// TIA Portal V17 export
// export: Created 2024-08-26T21:10:48.4510151Z, ExportSetting WithDefaults, DisplayName Totally Integrated Automation Portal, DisplayVersion V17 Update 7, DisplayName TIA Portal Openness, DisplayVersion V17 Update 7, DisplayName TIA Portal Version Control Interface, DisplayVersion V17, DisplayName SINAMICS Startdrive Advanced, DisplayVersion V17 SP2, DisplayName SINAMICS Startdrive G110M, G120, G120C, G120D, G120P, G115D, DisplayVersion V17 SP2, DisplayName SINAMICS Startdrive G130, G150, S120, S150, SINAMICS MV, S210, DisplayVersion V17 SP2, DisplayName STEP 7 Professional, DisplayVersion V17 Update 7, DisplayName STEP 7 Safety, DisplayVersion V17 Update 6, DisplayName WinCC Advanced / Unified PC, DisplayVersion V17 Update 7
FUNCTION "FC_EKS" : Void   // FC305, LAD
TITLE = Euchner Management EKS KEY
{ S7_Optimized_Access := 'FALSE' }
VERSION : 0.1
// stored: AutoNumber false, IsIECCheckEnabled false, SetENOAutomatically false, UDAEnableTagReadback false
   VAR_INPUT
      iKEY_IN : Bool;
      iEKS_LEVEL : Byte;
      iEKS_EMPLOYEE_ID : DWord;
      iEKS_KEY_ID1 : DWord;
      iEKS_KEY_ID2 : DWord;
      iEKS_JOB_FINISHED : Bool;
      "Current_page_of HMI" : Word;
   END_VAR
   VAR_OUTPUT
      qEKS_START_ADDRESS : Byte;
      qEKS_DATA_LENGTH : Byte;
      qEKS_DATA_1 : Byte;
      qEKS_DATA_2 : DWord;
      qEKS_WRITE_CMD : Bool;
   END_VAR
   VAR_TEMP
      tNone : Bool;
      tDBAddressKeys : Int;
      tDBAddressHMIPage : Int;
      tDBKeyStructLength : Int;
      tDBAddress : Int;
      tDBLength : Int;
      tCycle : Int;
      tFill : Int;
      tKey : "udt_EKS_KEY";
      tDBStartAddress : Int;
      tsearch : Bool;
      i : Int;
   END_VAR
   VAR CONSTANT
      DB : Byte := 16#84;
   END_VAR
   VAR_TEMP   // added for the SCL form of the ladder/FBD networks
      _w1 : Bool;
      _w2 : Bool;
   END_VAR
BEGIN

REGION Network 1: Actual HMI page index limits
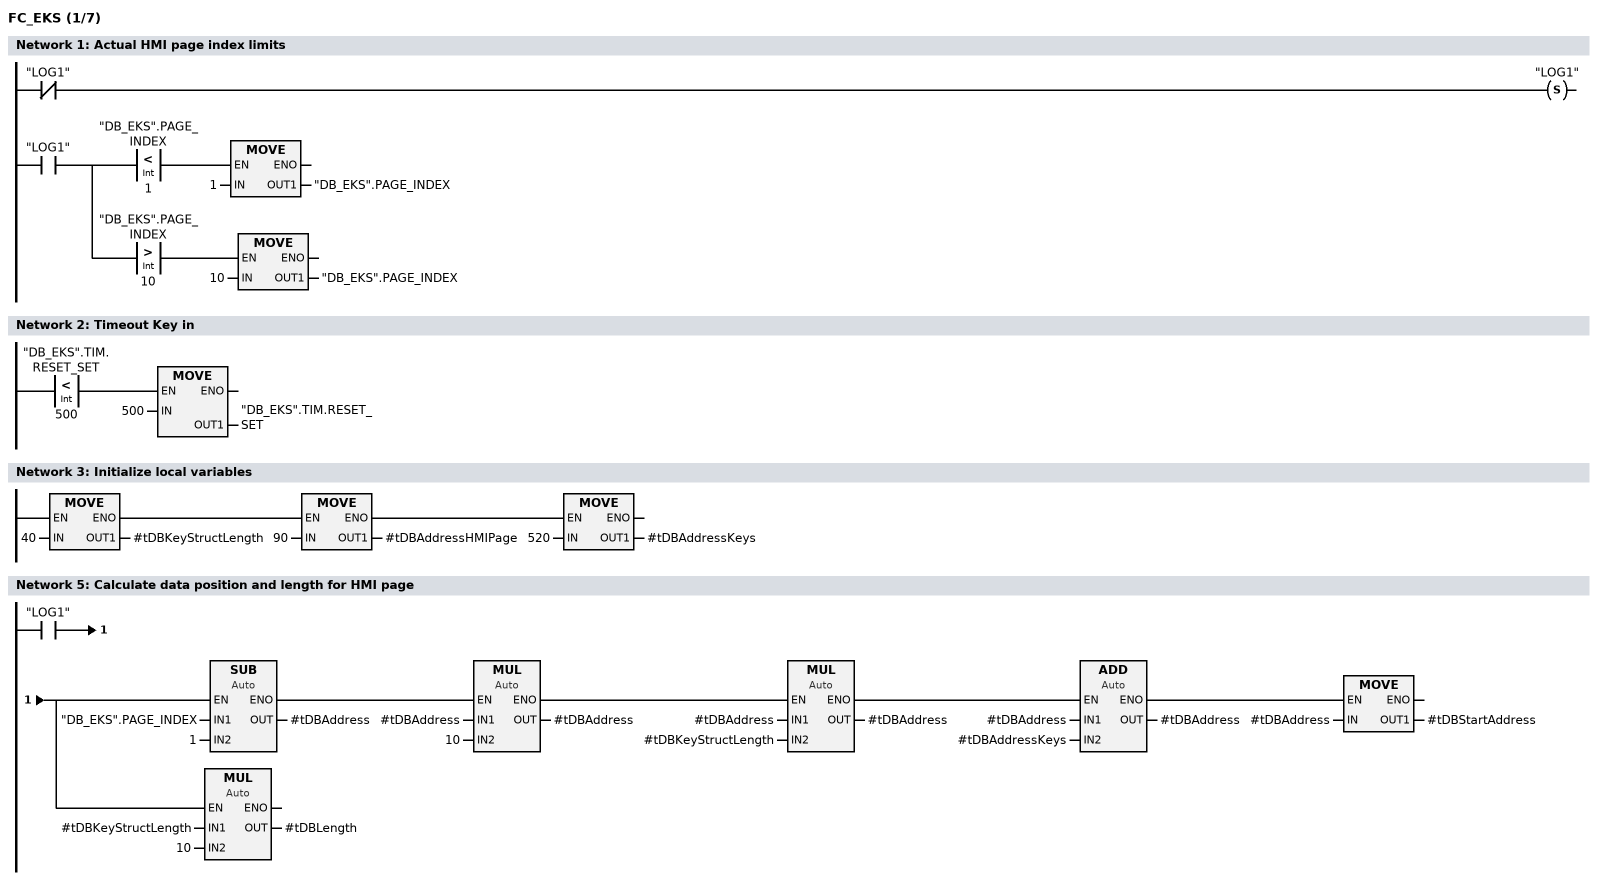
   RUNG wire#powerrail
      I_Contact( "LOG1" )
      S_Coil( "LOG1" )
   END_RUNG
   RUNG wire#powerrail
      Contact( "LOG1" )
      wire#w1
      { S7_Templates := "SrcType := Int" } LT_Contact(in1 := "DB_EKS".PAGE_INDEX, in2 := 1)
      Move(in := 1, out1 => "DB_EKS".PAGE_INDEX)
   END_RUNG
   RUNG wire#w1
      { S7_Templates := "SrcType := Int" } GT_Contact(in1 := "DB_EKS".PAGE_INDEX, in2 := 10)
      Move(in := 10, out1 => "DB_EKS".PAGE_INDEX)
   END_RUNG
   // the same network as SCL:
   IF NOT "LOG1" THEN "LOG1" := TRUE; END_IF;
   IF "LOG1" AND ("DB_EKS".PAGE_INDEX < 1) THEN "DB_EKS".PAGE_INDEX := 1; END_IF;
   IF "LOG1" AND ("DB_EKS".PAGE_INDEX > 10) THEN "DB_EKS".PAGE_INDEX := 10; END_IF;
END_REGION

REGION Network 2: Timeout Key in
   RUNG wire#powerrail
      { S7_Templates := "SrcType := Int" } LT_Contact(in1 := "DB_EKS".TIM.RESET_SET, in2 := 500)
      Move(in := 500, out1 => "DB_EKS".TIM.RESET_SET)
   END_RUNG
   // the same network as SCL:
   IF "DB_EKS".TIM.RESET_SET < 500 THEN "DB_EKS".TIM.RESET_SET := 500; END_IF;
END_REGION

REGION Network 3: Initialize local variables
   RUNG wire#powerrail
      Move(in := 40, out1 => #tDBKeyStructLength)
      Move(in := 90, out1 => #tDBAddressHMIPage)
      Move(in := 520, out1 => #tDBAddressKeys)
   END_RUNG
   // the same network as SCL:
   #tDBKeyStructLength := 40;
   #tDBAddressHMIPage := 90;
   #tDBAddressKeys := 520;
END_REGION

REGION Network 5: Calculate data position and length for HMI page
   RUNG wire#powerrail
      Contact( "LOG1" )
      wire#w1
      Sub(in1 := "DB_EKS".PAGE_INDEX, in2 := 1, out => #tDBAddress)
      Mul(in1 := #tDBAddress, in2 := 10, out => #tDBAddress)
      Mul(in1 := #tDBAddress, in2 := #tDBKeyStructLength, out => #tDBAddress)
      Add(in1 := #tDBAddress, in2 := #tDBAddressKeys, out => #tDBAddress)
      Move(in := #tDBAddress, out1 => #tDBStartAddress)
   END_RUNG
   RUNG wire#w1
      Mul(in1 := #tDBKeyStructLength, in2 := 10, out => #tDBLength)
   END_RUNG
   // the same network as SCL:
   IF "LOG1" THEN
       #tDBAddress := "DB_EKS".PAGE_INDEX - 1;
       #tDBAddress := #tDBAddress * 10;
       #tDBAddress := #tDBAddress * #tDBKeyStructLength;
       #tDBAddress := #tDBAddress + #tDBAddressKeys;
       #tDBStartAddress := #tDBAddress;
       #tDBLength := #tDBKeyStructLength * 10;
   END_IF;
END_REGION

REGION Network 6 (SCL): Copy data for page (10 keys)
   POKE_BLK(area_src:=#DB,
            dbNumber_src:=305,
            byteOffset_src:=#tDBAddress,
            area_dest:=#DB,
            dbNumber_dest:=305,
            byteOffset_dest:=90,
            count:=#tDBLength);
END_REGION

REGION Network 8: Inserted key
   // Store_Key_In is used to display only 1 time the level of euchner during storage function.
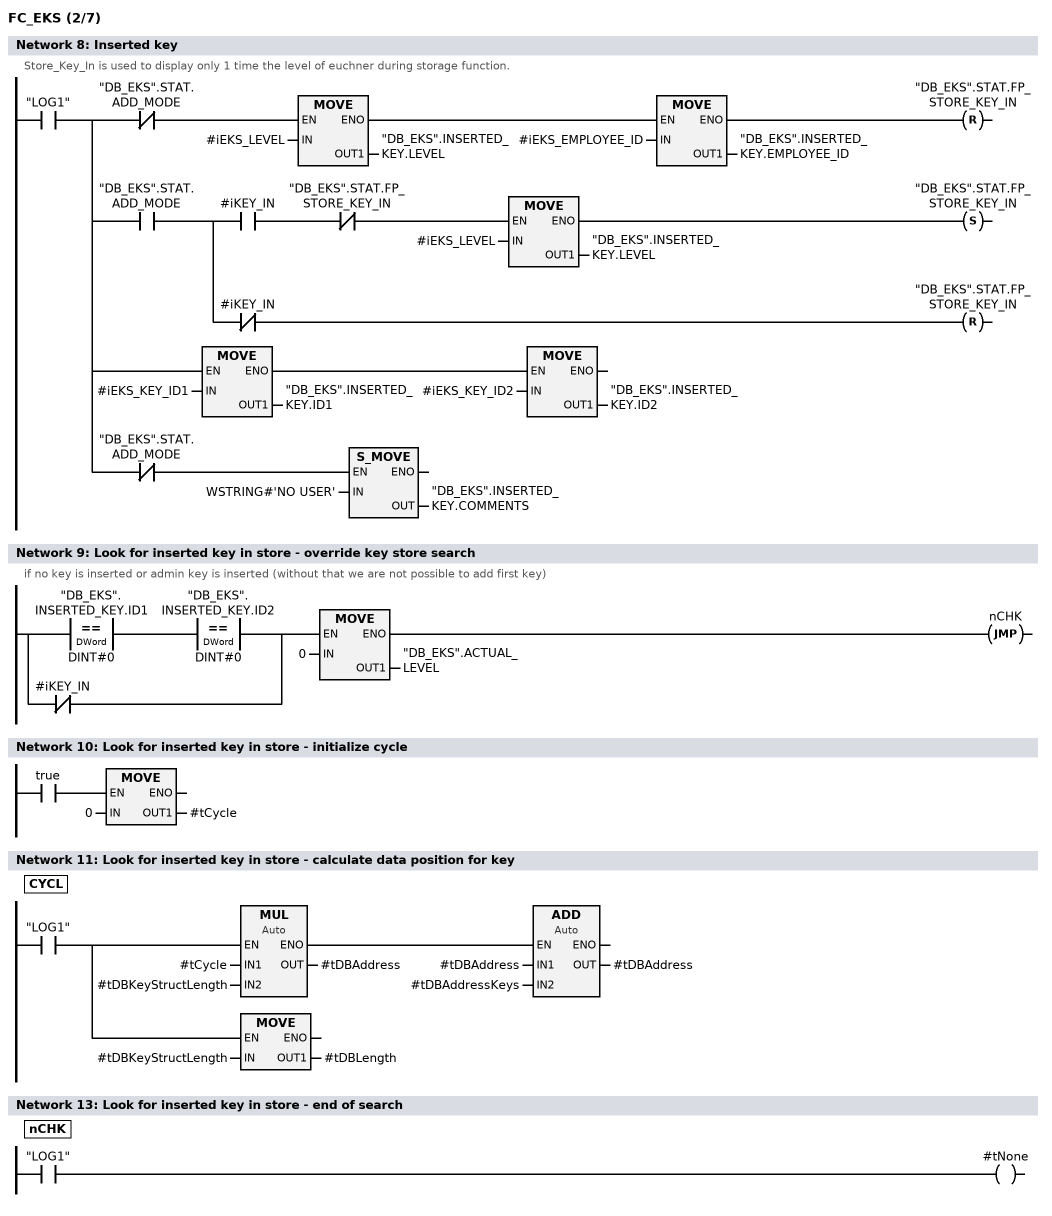
   RUNG wire#powerrail
      Contact( "LOG1" )
      wire#w1
      I_Contact( "DB_EKS".STAT.ADD_MODE )
      Move(in := #iEKS_LEVEL, out1 => "DB_EKS".INSERTED_KEY.LEVEL)
      Move(in := #iEKS_EMPLOYEE_ID, out1 => "DB_EKS".INSERTED_KEY.EMPLOYEE_ID)
      R_Coil( "DB_EKS".STAT.FP_STORE_KEY_IN )
   END_RUNG
   RUNG wire#w1
      Contact( "DB_EKS".STAT.ADD_MODE )
      wire#w2
      Contact( #iKEY_IN )
      I_Contact( "DB_EKS".STAT.FP_STORE_KEY_IN )
      Move(in := #iEKS_LEVEL, out1 => "DB_EKS".INSERTED_KEY.LEVEL)
      S_Coil( "DB_EKS".STAT.FP_STORE_KEY_IN )
   END_RUNG
   RUNG wire#w2
      I_Contact( #iKEY_IN )
      R_Coil( "DB_EKS".STAT.FP_STORE_KEY_IN )
   END_RUNG
   RUNG wire#w1
      Move(in := #iEKS_KEY_ID1, out1 => "DB_EKS".INSERTED_KEY.ID1)
      Move(in := #iEKS_KEY_ID2, out1 => "DB_EKS".INSERTED_KEY.ID2)
   END_RUNG
   RUNG wire#w1
      I_Contact( "DB_EKS".STAT.ADD_MODE )
      S_Move(in := WSTRING#'NO USER', out => "DB_EKS".INSERTED_KEY.COMMENTS)
   END_RUNG
   // the same network as SCL:
   IF "LOG1" AND NOT "DB_EKS".STAT.ADD_MODE THEN
       "DB_EKS".INSERTED_KEY.LEVEL := #iEKS_LEVEL;
       "DB_EKS".INSERTED_KEY.EMPLOYEE_ID := #iEKS_EMPLOYEE_ID;
       "DB_EKS".STAT.FP_STORE_KEY_IN := FALSE;
   END_IF;
   #_w1 := "LOG1" AND "DB_EKS".STAT.ADD_MODE;
   IF #_w1 AND #iKEY_IN AND NOT "DB_EKS".STAT.FP_STORE_KEY_IN THEN
       "DB_EKS".INSERTED_KEY.LEVEL := #iEKS_LEVEL;
       "DB_EKS".STAT.FP_STORE_KEY_IN := TRUE;
   END_IF;
   IF #_w1 AND NOT #iKEY_IN THEN "DB_EKS".STAT.FP_STORE_KEY_IN := FALSE; END_IF;
   IF "LOG1" THEN
       "DB_EKS".INSERTED_KEY.ID1 := #iEKS_KEY_ID1;
       "DB_EKS".INSERTED_KEY.ID2 := #iEKS_KEY_ID2;
   END_IF;
   IF "LOG1" AND NOT "DB_EKS".STAT.ADD_MODE THEN "DB_EKS".INSERTED_KEY.COMMENTS := WSTRING#'NO USER'; END_IF;
END_REGION

REGION Network 9: Look for inserted key in store - override key store search
   // if no key is inserted or admin key is inserted (without that we are not possible to add first key)
   RUNG wire#powerrail
      { S7_Templates := "SrcType := DWord" } EQ_Contact(in1 := "DB_EKS".INSERTED_KEY.ID1, in2 := DINT#0)
      { S7_Templates := "SrcType := DWord" } EQ_Contact(in1 := "DB_EKS".INSERTED_KEY.ID2, in2 := DINT#0)
      wire#w1
      Move(in := 0, out1 => "DB_EKS".ACTUAL_LEVEL)
      JumpCoil( nCHK )
   END_RUNG
   RUNG wire#powerrail
      I_Contact( #iKEY_IN )
   END_RUNG wire#w1
   // the same network as SCL:
   #_w1 := (("DB_EKS".INSERTED_KEY.ID1 = DINT#0) AND ("DB_EKS".INSERTED_KEY.ID2 = DINT#0)) OR NOT #iKEY_IN;
   IF #_w1 THEN
       "DB_EKS".ACTUAL_LEVEL := 0;
       GOTO nCHK;
   END_IF;
END_REGION

REGION Network 10: Look for inserted key in store - initialize cycle
   RUNG wire#powerrail
      Contact( true )
      Move(in := 0, out1 => #tCycle)
   END_RUNG
   // the same network as SCL:
   IF true THEN #tCycle := 0; END_IF;
END_REGION

REGION Network 11: Look for inserted key in store - calculate data position for key
   Label( CYCL )
   RUNG wire#powerrail
      Contact( "LOG1" )
      wire#w1
      Mul(in1 := #tCycle, in2 := #tDBKeyStructLength, out => #tDBAddress)
      Add(in1 := #tDBAddress, in2 := #tDBAddressKeys, out => #tDBAddress)
   END_RUNG
   RUNG wire#w1
      Move(in := #tDBKeyStructLength, out1 => #tDBLength)
   END_RUNG
   // the same network as SCL:
   CYCL:
   IF "LOG1" THEN
       #tDBAddress := #tCycle * #tDBKeyStructLength;
       #tDBAddress := #tDBAddress + #tDBAddressKeys;
       #tDBLength := #tDBKeyStructLength;
   END_IF;
END_REGION

REGION Network 12 (SCL): Look for inserted key in store - check ID of stored key
   FOR #i := 1 TO 130 DO
       #tKey := "DB_EKS".KEYS[#i];
       IF (#tKey.ID1 = "DB_EKS".INSERTED_KEY.ID1) AND
           (#tKey.ID2 = "DB_EKS".INSERTED_KEY.ID2) THEN
           "DB_EKS".ACTUAL_LEVEL := #tKey.LEVEL;
           "DB_EKS".INSERTED_KEY.COMMENTS := #tKey.COMMENTS;
           EXIT;
       END_IF;
   END_FOR;
END_REGION

REGION Network 13: Look for inserted key in store - end of search
   Label( nCHK )
   RUNG wire#powerrail
      Contact( "LOG1" )
      Coil( #tNone )
   END_RUNG
   // the same network as SCL:
   nCHK:
   #tNone := "LOG1";
END_REGION

REGION Network 14: Reset of EKS higher levels until key is removed
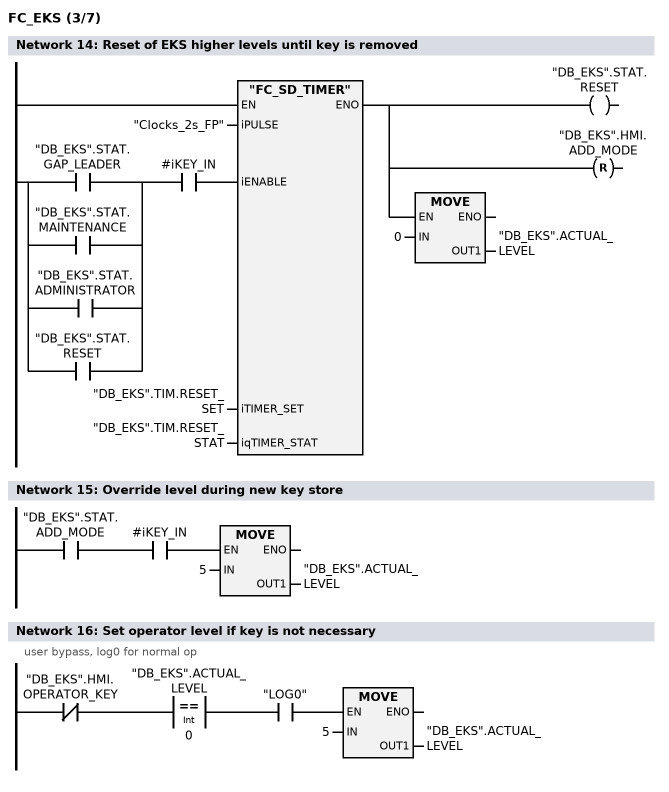
   RUNG wire#powerrail
      "FC_SD_TIMER"(iENABLE := wire#w2, iPULSE := "Clocks_2s_FP", iTIMER_SET := "DB_EKS".TIM.RESET_SET, iqTIMER_STAT := "DB_EKS".TIM.RESET_STAT)
      wire#w3
      Coil( "DB_EKS".STAT.RESET )
   END_RUNG
   RUNG wire#powerrail
      Contact( "DB_EKS".STAT.GAP_LEADER )
      wire#w1
      Contact( #iKEY_IN )
   END_RUNG wire#w2
   RUNG wire#powerrail
      Contact( "DB_EKS".STAT.MAINTENANCE )
   END_RUNG wire#w1
   RUNG wire#powerrail
      Contact( "DB_EKS".STAT.ADMINISTRATOR )
   END_RUNG wire#w1
   RUNG wire#powerrail
      Contact( "DB_EKS".STAT.RESET )
   END_RUNG wire#w1
   RUNG wire#w3
      R_Coil( "DB_EKS".HMI.ADD_MODE )
   END_RUNG
   RUNG wire#w3
      Move(in := 0, out1 => "DB_EKS".ACTUAL_LEVEL)
   END_RUNG
   // the same network as SCL:
   "FC_SD_TIMER"(iPULSE := "Clocks_2s_FP",
                 iENABLE := ("DB_EKS".STAT.GAP_LEADER OR "DB_EKS".STAT.MAINTENANCE OR "DB_EKS".STAT.ADMINISTRATOR OR "DB_EKS".STAT.RESET) AND #iKEY_IN,
                 iTIMER_SET := "DB_EKS".TIM.RESET_SET,
                 iqTIMER_STAT := "DB_EKS".TIM.RESET_STAT,
                 ENO => #_w1);
   "DB_EKS".STAT.RESET := #_w1;
   IF #_w1 THEN
       "DB_EKS".HMI.ADD_MODE := FALSE;
       "DB_EKS".ACTUAL_LEVEL := 0;
   END_IF;
END_REGION

REGION Network 15: Override level during new key store
   RUNG wire#powerrail
      Contact( "DB_EKS".STAT.ADD_MODE )
      Contact( #iKEY_IN )
      Move(in := 5, out1 => "DB_EKS".ACTUAL_LEVEL)
   END_RUNG
   // the same network as SCL:
   IF "DB_EKS".STAT.ADD_MODE AND #iKEY_IN THEN "DB_EKS".ACTUAL_LEVEL := 5; END_IF;
END_REGION

REGION Network 16: Set operator level if key is not necessary
   // user bypass, log0 for normal op
   RUNG wire#powerrail
      I_Contact( "DB_EKS".HMI.OPERATOR_KEY )
      { S7_Templates := "SrcType := Int" } EQ_Contact(in1 := "DB_EKS".ACTUAL_LEVEL, in2 := 0)
      Contact( "LOG0" )
      Move(in := 5, out1 => "DB_EKS".ACTUAL_LEVEL)
   END_RUNG
   // the same network as SCL:
   IF NOT "DB_EKS".HMI.OPERATOR_KEY AND ("DB_EKS".ACTUAL_LEVEL = 0) AND "LOG0" THEN
       "DB_EKS".ACTUAL_LEVEL := 5;
   END_IF;
END_REGION

REGION Network 17: EKS levels
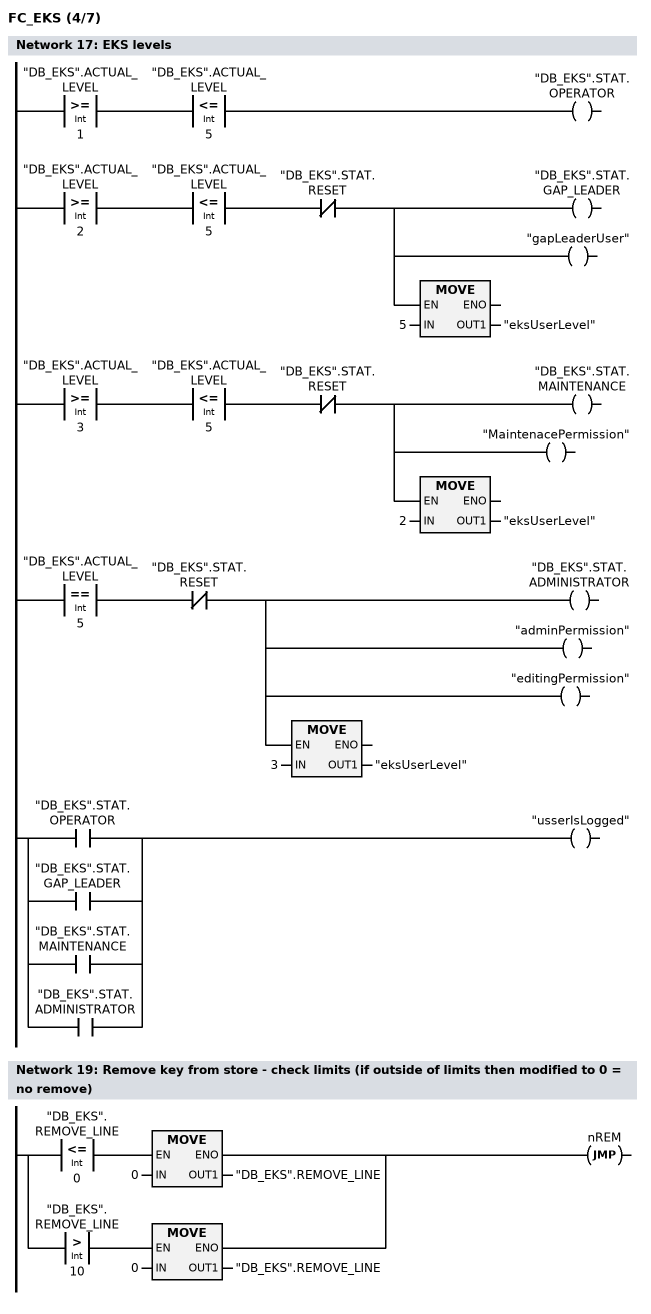
   RUNG wire#powerrail
      { S7_Templates := "SrcType := Int" } GE_Contact(in1 := "DB_EKS".ACTUAL_LEVEL, in2 := 1)
      { S7_Templates := "SrcType := Int" } LE_Contact(in1 := "DB_EKS".ACTUAL_LEVEL, in2 := 5)
      Coil( "DB_EKS".STAT.OPERATOR )
   END_RUNG
   RUNG wire#powerrail
      { S7_Templates := "SrcType := Int" } GE_Contact(in1 := "DB_EKS".ACTUAL_LEVEL, in2 := 2)
      { S7_Templates := "SrcType := Int" } LE_Contact(in1 := "DB_EKS".ACTUAL_LEVEL, in2 := 5)
      I_Contact( "DB_EKS".STAT.RESET )
      wire#w1
      Coil( "DB_EKS".STAT.GAP_LEADER )
   END_RUNG
   RUNG wire#w1
      Coil( "gapLeaderUser" )
   END_RUNG
   RUNG wire#w1
      Move(in := 5, out1 => "eksUserLevel")
   END_RUNG
   RUNG wire#powerrail
      { S7_Templates := "SrcType := Int" } GE_Contact(in1 := "DB_EKS".ACTUAL_LEVEL, in2 := 3)
      { S7_Templates := "SrcType := Int" } LE_Contact(in1 := "DB_EKS".ACTUAL_LEVEL, in2 := 5)
      I_Contact( "DB_EKS".STAT.RESET )
      wire#w2
      Coil( "DB_EKS".STAT.MAINTENANCE )
   END_RUNG
   RUNG wire#w2
      Coil( "MaintenacePermission" )
   END_RUNG
   RUNG wire#w2
      Move(in := 2, out1 => "eksUserLevel")
   END_RUNG
   RUNG wire#powerrail
      { S7_Templates := "SrcType := Int" } EQ_Contact(in1 := "DB_EKS".ACTUAL_LEVEL, in2 := 5)
      I_Contact( "DB_EKS".STAT.RESET )
      wire#w3
      Coil( "DB_EKS".STAT.ADMINISTRATOR )
   END_RUNG
   RUNG wire#w3
      Coil( "adminPermission" )
   END_RUNG
   RUNG wire#w3
      Coil( "editingPermission" )
   END_RUNG
   RUNG wire#w3
      Move(in := 3, out1 => "eksUserLevel")
   END_RUNG
   RUNG wire#powerrail
      Contact( "DB_EKS".STAT.OPERATOR )
      wire#w4
      Coil( "usserIsLogged" )
   END_RUNG
   RUNG wire#powerrail
      Contact( "DB_EKS".STAT.GAP_LEADER )
   END_RUNG wire#w4
   RUNG wire#powerrail
      Contact( "DB_EKS".STAT.MAINTENANCE )
   END_RUNG wire#w4
   RUNG wire#powerrail
      Contact( "DB_EKS".STAT.ADMINISTRATOR )
   END_RUNG wire#w4
   // the same network as SCL:
   "DB_EKS".STAT.OPERATOR := ("DB_EKS".ACTUAL_LEVEL >= 1) AND ("DB_EKS".ACTUAL_LEVEL <= 5);
   "DB_EKS".STAT.GAP_LEADER := ("DB_EKS".ACTUAL_LEVEL >= 2) AND ("DB_EKS".ACTUAL_LEVEL <= 5) AND NOT "DB_EKS".STAT.RESET;
   "gapLeaderUser" := "DB_EKS".STAT.GAP_LEADER;
   IF "DB_EKS".STAT.GAP_LEADER THEN "eksUserLevel" := 5; END_IF;
   "DB_EKS".STAT.MAINTENANCE := ("DB_EKS".ACTUAL_LEVEL >= 3) AND ("DB_EKS".ACTUAL_LEVEL <= 5) AND NOT "DB_EKS".STAT.RESET;
   "MaintenacePermission" := "DB_EKS".STAT.MAINTENANCE;
   IF "DB_EKS".STAT.MAINTENANCE THEN "eksUserLevel" := 2; END_IF;
   "DB_EKS".STAT.ADMINISTRATOR := ("DB_EKS".ACTUAL_LEVEL = 5) AND NOT "DB_EKS".STAT.RESET;
   "adminPermission" := "DB_EKS".STAT.ADMINISTRATOR;
   "editingPermission" := "DB_EKS".STAT.ADMINISTRATOR;
   IF "DB_EKS".STAT.ADMINISTRATOR THEN "eksUserLevel" := 3; END_IF;
   "usserIsLogged" := "DB_EKS".STAT.OPERATOR OR "DB_EKS".STAT.GAP_LEADER OR "DB_EKS".STAT.MAINTENANCE OR "DB_EKS".STAT.ADMINISTRATOR;
END_REGION

REGION Network 19: Remove key from store - check limits (if outside of limits then modified to 0 = no remove)
   RUNG wire#powerrail
      { S7_Templates := "SrcType := Int" } LE_Contact(in1 := "DB_EKS".REMOVE_LINE, in2 := 0)
      Move(in := 0, out1 => "DB_EKS".REMOVE_LINE)
      wire#w1
      JumpCoil( nREM )
   END_RUNG
   RUNG wire#powerrail
      { S7_Templates := "SrcType := Int" } GT_Contact(in1 := "DB_EKS".REMOVE_LINE, in2 := 10)
      Move(in := 0, out1 => "DB_EKS".REMOVE_LINE)
   END_RUNG wire#w1
   // the same network as SCL:
   #_w1 := "DB_EKS".REMOVE_LINE <= 0;
   IF #_w1 THEN "DB_EKS".REMOVE_LINE := 0; END_IF;
   #_w2 := "DB_EKS".REMOVE_LINE > 10;
   IF #_w2 THEN "DB_EKS".REMOVE_LINE := 0; END_IF;
   IF #_w1 OR #_w2 THEN GOTO nREM; END_IF;
END_REGION

REGION Network 20: Remove key from store - calculate data position and length for HMI page
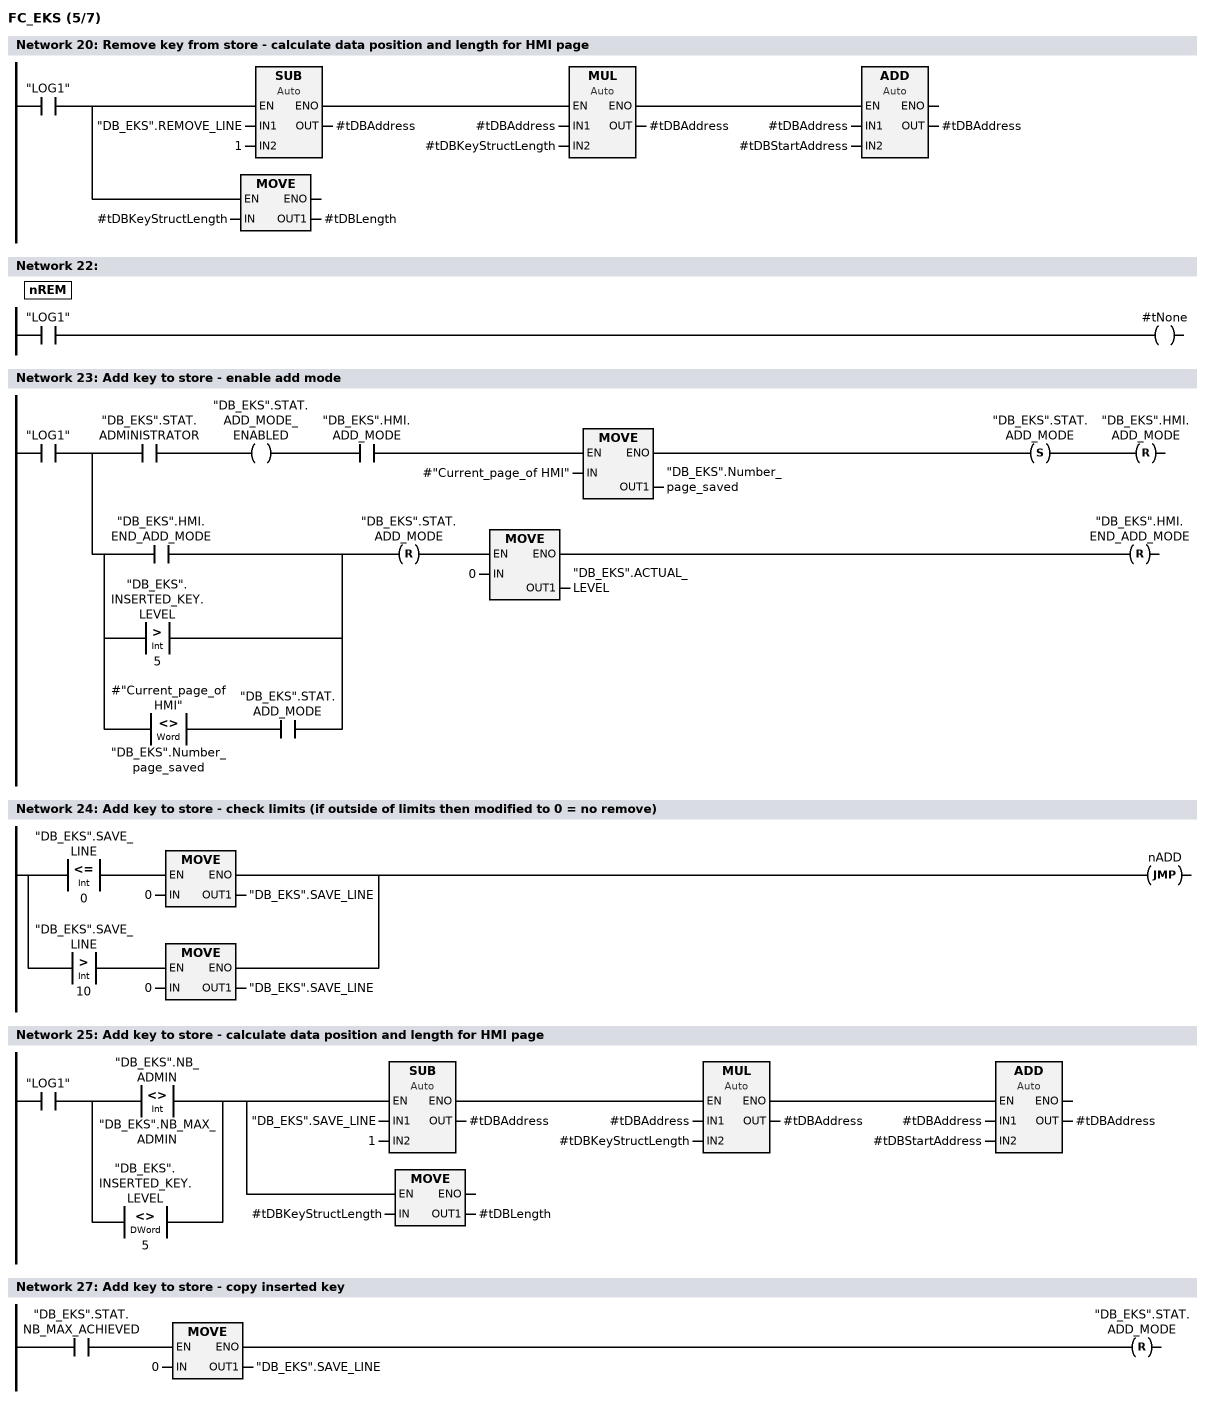
   RUNG wire#powerrail
      Contact( "LOG1" )
      wire#w1
      Sub(in1 := "DB_EKS".REMOVE_LINE, in2 := 1, out => #tDBAddress)
      Mul(in1 := #tDBAddress, in2 := #tDBKeyStructLength, out => #tDBAddress)
      Add(in1 := #tDBAddress, in2 := #tDBStartAddress, out => #tDBAddress)
   END_RUNG
   RUNG wire#w1
      Move(in := #tDBKeyStructLength, out1 => #tDBLength)
   END_RUNG
   // the same network as SCL:
   IF "LOG1" THEN
       #tDBAddress := "DB_EKS".REMOVE_LINE - 1;
       #tDBAddress := #tDBAddress * #tDBKeyStructLength;
       #tDBAddress := #tDBAddress + #tDBStartAddress;
       #tDBLength := #tDBKeyStructLength;
   END_IF;
END_REGION

REGION Network 21 (SCL): Remove key from store - delete key
   #tFill := 0;

   POKE_BLK(area_src:=#DB,
            dbNumber_src:=305,
            byteOffset_src:=5720,
            area_dest:=#DB,
            dbNumber_dest:=305,
            byteOffset_dest:=#tDBAddress,
            count:=#tDBLength);

   "DB_EKS".REMOVE_LINE := 0;
END_REGION

REGION Network 22
   Label( nREM )
   RUNG wire#powerrail
      Contact( "LOG1" )
      Coil( #tNone )
   END_RUNG
   // the same network as SCL:
   nREM:
   #tNone := "LOG1";
END_REGION

REGION Network 23: Add key to store - enable add mode
   RUNG wire#powerrail
      Contact( "LOG1" )
      wire#w1
      Contact( "DB_EKS".STAT.ADMINISTRATOR )
      Coil( "DB_EKS".STAT.ADD_MODE_ENABLED )
      Contact( "DB_EKS".HMI.ADD_MODE )
      Move(in := #"Current_page_of HMI", out1 => "DB_EKS".Number_page_saved)
      S_Coil( "DB_EKS".STAT.ADD_MODE )
      R_Coil( "DB_EKS".HMI.ADD_MODE )
   END_RUNG
   RUNG wire#w1
      Contact( "DB_EKS".HMI.END_ADD_MODE )
      wire#w2
      R_Coil( "DB_EKS".STAT.ADD_MODE )
      Move(in := 0, out1 => "DB_EKS".ACTUAL_LEVEL)
      R_Coil( "DB_EKS".HMI.END_ADD_MODE )
   END_RUNG
   RUNG wire#w1
      { S7_Templates := "SrcType := Int" } GT_Contact(in1 := "DB_EKS".INSERTED_KEY.LEVEL, in2 := 5)
   END_RUNG wire#w2
   RUNG wire#w1
      { S7_Templates := "SrcType := Word" } NE_Contact(in1 := #"Current_page_of HMI", in2 := "DB_EKS".Number_page_saved)
      Contact( "DB_EKS".STAT.ADD_MODE )
   END_RUNG wire#w2
   // the same network as SCL:
   "DB_EKS".STAT.ADD_MODE_ENABLED := "LOG1" AND "DB_EKS".STAT.ADMINISTRATOR;
   IF "DB_EKS".STAT.ADD_MODE_ENABLED AND "DB_EKS".HMI.ADD_MODE THEN
       "DB_EKS".Number_page_saved := #"Current_page_of HMI";
       "DB_EKS".STAT.ADD_MODE := TRUE;
       "DB_EKS".HMI.ADD_MODE := FALSE;
   END_IF;
   #_w1 := "LOG1" AND ("DB_EKS".HMI.END_ADD_MODE OR ("DB_EKS".INSERTED_KEY.LEVEL > 5) OR ((#"Current_page_of HMI" <> "DB_EKS".Number_page_saved) AND "DB_EKS".STAT.ADD_MODE));
   IF #_w1 THEN
       "DB_EKS".STAT.ADD_MODE := FALSE;
       "DB_EKS".ACTUAL_LEVEL := 0;
       "DB_EKS".HMI.END_ADD_MODE := FALSE;
   END_IF;
END_REGION

REGION Network 24: Add key to store - check limits (if outside of limits then modified to 0 = no remove)
   RUNG wire#powerrail
      { S7_Templates := "SrcType := Int" } LE_Contact(in1 := "DB_EKS".SAVE_LINE, in2 := 0)
      Move(in := 0, out1 => "DB_EKS".SAVE_LINE)
      wire#w1
      JumpCoil( nADD )
   END_RUNG
   RUNG wire#powerrail
      { S7_Templates := "SrcType := Int" } GT_Contact(in1 := "DB_EKS".SAVE_LINE, in2 := 10)
      Move(in := 0, out1 => "DB_EKS".SAVE_LINE)
   END_RUNG wire#w1
   // the same network as SCL:
   #_w1 := "DB_EKS".SAVE_LINE <= 0;
   IF #_w1 THEN "DB_EKS".SAVE_LINE := 0; END_IF;
   #_w2 := "DB_EKS".SAVE_LINE > 10;
   IF #_w2 THEN "DB_EKS".SAVE_LINE := 0; END_IF;
   IF #_w1 OR #_w2 THEN GOTO nADD; END_IF;
END_REGION

REGION Network 25: Add key to store - calculate data position and length for HMI page
   RUNG wire#powerrail
      Contact( "LOG1" )
      wire#w1
      { S7_Templates := "SrcType := Int" } NE_Contact(in1 := "DB_EKS".NB_ADMIN, in2 := "DB_EKS".NB_MAX_ADMIN)
      wire#w2
      Sub(in1 := "DB_EKS".SAVE_LINE, in2 := 1, out => #tDBAddress)
      Mul(in1 := #tDBAddress, in2 := #tDBKeyStructLength, out => #tDBAddress)
      Add(in1 := #tDBAddress, in2 := #tDBStartAddress, out => #tDBAddress)
   END_RUNG
   RUNG wire#w1
      { S7_Templates := "SrcType := DWord" } NE_Contact(in1 := "DB_EKS".INSERTED_KEY.LEVEL, in2 := 5)
   END_RUNG wire#w2
   RUNG wire#w2
      Move(in := #tDBKeyStructLength, out1 => #tDBLength)
   END_RUNG
   // the same network as SCL:
   IF "LOG1" AND (("DB_EKS".NB_ADMIN <> "DB_EKS".NB_MAX_ADMIN) OR ("DB_EKS".INSERTED_KEY.LEVEL <> 5)) THEN
       #tDBAddress := "DB_EKS".SAVE_LINE - 1;
       #tDBAddress := #tDBAddress * #tDBKeyStructLength;
       #tDBAddress := #tDBAddress + #tDBStartAddress;
       #tDBLength := #tDBKeyStructLength;
   END_IF;
END_REGION

REGION Network 26 (SCL): Add key to store - copy inserted key
   IF ("DB_EKS".INSERTED_KEY.LEVEL = 5  & NOT "DB_EKS".STAT.NB_MAX_ACHIEVED) OR
       ("DB_EKS".INSERTED_KEY.LEVEL <> 5) THEN
       POKE_BLK(area_src := #DB,
                dbNumber_src := 305,
                byteOffset_src := 50,
                area_dest := #DB,
                dbNumber_dest := 305,
                byteOffset_dest := #tDBAddress,
                count := #tDBLength);
      "DB_EKS".SAVE_LINE := 0;
   END_IF;
END_REGION

REGION Network 27: Add key to store - copy inserted key
   RUNG wire#powerrail
      Contact( "DB_EKS".STAT.NB_MAX_ACHIEVED )
      Move(in := 0, out1 => "DB_EKS".SAVE_LINE)
      R_Coil( "DB_EKS".STAT.ADD_MODE )
   END_RUNG
   // the same network as SCL:
   IF "DB_EKS".STAT.NB_MAX_ACHIEVED THEN
       "DB_EKS".SAVE_LINE := 0;
       "DB_EKS".STAT.ADD_MODE := FALSE;
   END_IF;
END_REGION

REGION Network 28
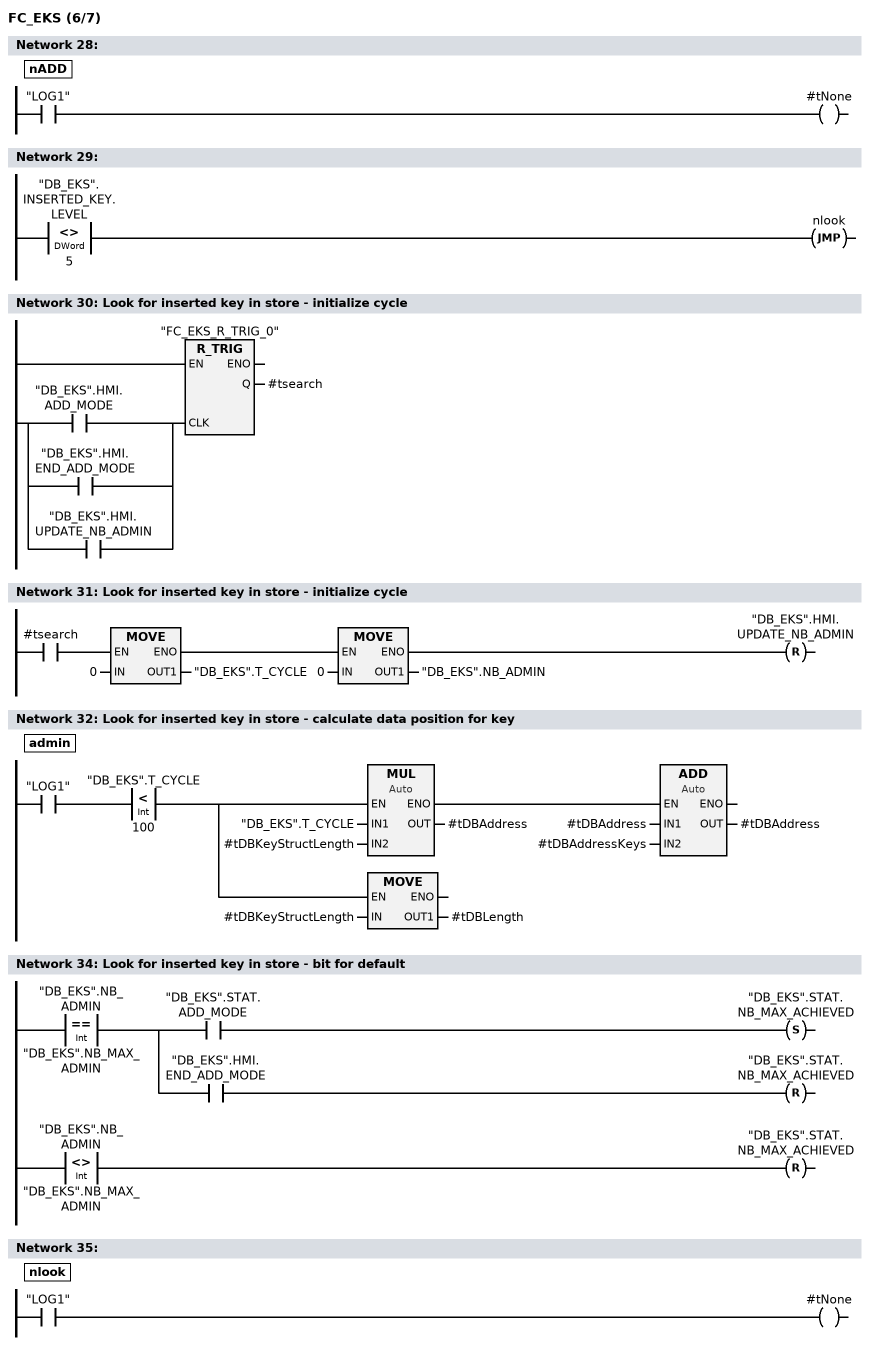
   Label( nADD )
   RUNG wire#powerrail
      Contact( "LOG1" )
      Coil( #tNone )
   END_RUNG
   // the same network as SCL:
   nADD:
   #tNone := "LOG1";
END_REGION

REGION Network 29
   RUNG wire#powerrail
      { S7_Templates := "SrcType := DWord" } NE_Contact(in1 := "DB_EKS".INSERTED_KEY.LEVEL, in2 := 5)
      JumpCoil( nlook )
   END_RUNG
   // the same network as SCL:
   IF "DB_EKS".INSERTED_KEY.LEVEL <> 5 THEN GOTO nlook; END_IF;
END_REGION

REGION Network 30: Look for inserted key in store - initialize cycle
   RUNG wire#powerrail
      "FC_EKS_R_TRIG_0".R_TRIG(CLK := wire#w1, Q => #tsearch)
   END_RUNG
   RUNG wire#powerrail
      Contact( "DB_EKS".HMI.ADD_MODE )
   END_RUNG wire#w1
   RUNG wire#powerrail
      Contact( "DB_EKS".HMI.END_ADD_MODE )
   END_RUNG wire#w1
   RUNG wire#powerrail
      Contact( "DB_EKS".HMI.UPDATE_NB_ADMIN )
   END_RUNG wire#w1
   // the same network as SCL:
   "FC_EKS_R_TRIG_0"(CLK := "DB_EKS".HMI.ADD_MODE OR "DB_EKS".HMI.END_ADD_MODE OR "DB_EKS".HMI.UPDATE_NB_ADMIN,   // R_TRIG
                     Q => #tsearch);
END_REGION

REGION Network 31: Look for inserted key in store - initialize cycle
   RUNG wire#powerrail
      Contact( #tsearch )
      Move(in := 0, out1 => "DB_EKS".T_CYCLE)
      Move(in := 0, out1 => "DB_EKS".NB_ADMIN)
      R_Coil( "DB_EKS".HMI.UPDATE_NB_ADMIN )
   END_RUNG
   // the same network as SCL:
   IF #tsearch THEN
       "DB_EKS".T_CYCLE := 0;
       "DB_EKS".NB_ADMIN := 0;
       "DB_EKS".HMI.UPDATE_NB_ADMIN := FALSE;
   END_IF;
END_REGION

REGION Network 32: Look for inserted key in store - calculate data position for key
   Label( admin )
   RUNG wire#powerrail
      Contact( "LOG1" )
      { S7_Templates := "SrcType := Int" } LT_Contact(in1 := "DB_EKS".T_CYCLE, in2 := 100)
      wire#w1
      Mul(in1 := "DB_EKS".T_CYCLE, in2 := #tDBKeyStructLength, out => #tDBAddress)
      Add(in1 := #tDBAddress, in2 := #tDBAddressKeys, out => #tDBAddress)
   END_RUNG
   RUNG wire#w1
      Move(in := #tDBKeyStructLength, out1 => #tDBLength)
   END_RUNG
   // the same network as SCL:
   admin:
   IF "LOG1" AND ("DB_EKS".T_CYCLE < 100) THEN
       #tDBAddress := "DB_EKS".T_CYCLE * #tDBKeyStructLength;
       #tDBAddress := #tDBAddress + #tDBAddressKeys;
       #tDBLength := #tDBKeyStructLength;
   END_IF;
END_REGION

REGION Network 33 (SCL): Look for inserted key in store - check ID of stored key
   FOR #i := 1 TO 100 DO
       #tKey := "DB_EKS".KEYS[#i];
       IF #tKey.LEVEL = 5 THEN
           "DB_EKS".NB_ADMIN += 1;
           CONTINUE;
       END_IF;
   END_FOR;
END_REGION

REGION Network 34: Look for inserted key in store - bit for default
   RUNG wire#powerrail
      { S7_Templates := "SrcType := Int" } EQ_Contact(in1 := "DB_EKS".NB_ADMIN, in2 := "DB_EKS".NB_MAX_ADMIN)
      wire#w1
      Contact( "DB_EKS".STAT.ADD_MODE )
      S_Coil( "DB_EKS".STAT.NB_MAX_ACHIEVED )
   END_RUNG
   RUNG wire#w1
      Contact( "DB_EKS".HMI.END_ADD_MODE )
      R_Coil( "DB_EKS".STAT.NB_MAX_ACHIEVED )
   END_RUNG
   RUNG wire#powerrail
      { S7_Templates := "SrcType := Int" } NE_Contact(in1 := "DB_EKS".NB_ADMIN, in2 := "DB_EKS".NB_MAX_ADMIN)
      R_Coil( "DB_EKS".STAT.NB_MAX_ACHIEVED )
   END_RUNG
   // the same network as SCL:
   #_w1 := "DB_EKS".NB_ADMIN = "DB_EKS".NB_MAX_ADMIN;
   IF #_w1 AND "DB_EKS".STAT.ADD_MODE THEN "DB_EKS".STAT.NB_MAX_ACHIEVED := TRUE; END_IF;
   IF #_w1 AND "DB_EKS".HMI.END_ADD_MODE THEN "DB_EKS".STAT.NB_MAX_ACHIEVED := FALSE; END_IF;
   IF "DB_EKS".NB_ADMIN <> "DB_EKS".NB_MAX_ADMIN THEN "DB_EKS".STAT.NB_MAX_ACHIEVED := FALSE; END_IF;
END_REGION

REGION Network 35
   Label( nlook )
   RUNG wire#powerrail
      Contact( "LOG1" )
      Coil( #tNone )
   END_RUNG
   // the same network as SCL:
   nlook:
   #tNone := "LOG1";
END_REGION

REGION Network 36: Write Level and Employer ID on Key
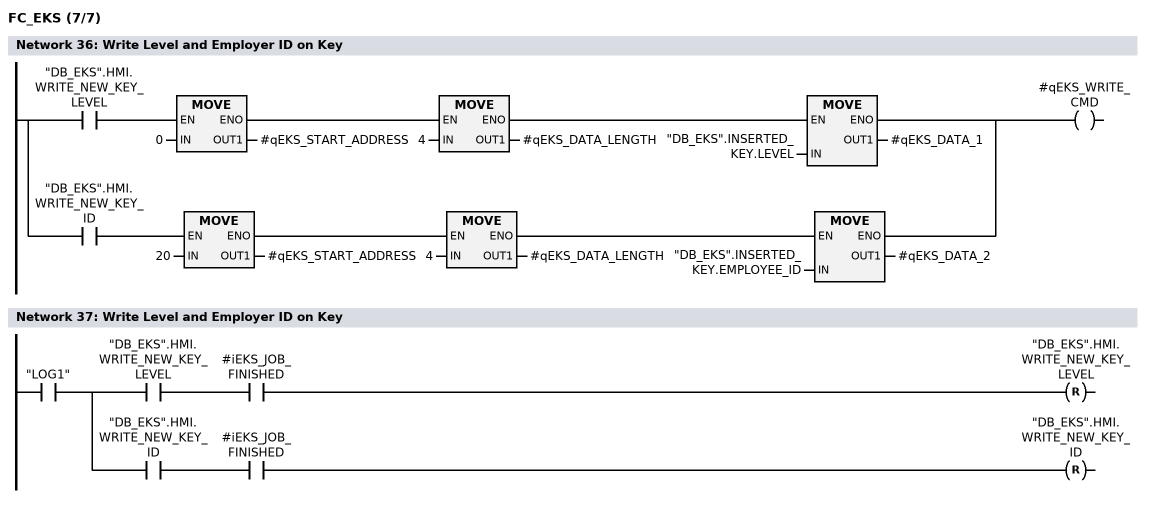
   RUNG wire#powerrail
      Contact( "DB_EKS".HMI.WRITE_NEW_KEY_LEVEL )
      Move(in := 0, out1 => #qEKS_START_ADDRESS)
      Move(in := 4, out1 => #qEKS_DATA_LENGTH)
      Move(in := "DB_EKS".INSERTED_KEY.LEVEL, out1 => #qEKS_DATA_1)
      wire#w1
      Coil( #qEKS_WRITE_CMD )
   END_RUNG
   RUNG wire#powerrail
      Contact( "DB_EKS".HMI.WRITE_NEW_KEY_ID )
      Move(in := 20, out1 => #qEKS_START_ADDRESS)
      Move(in := 4, out1 => #qEKS_DATA_LENGTH)
      Move(in := "DB_EKS".INSERTED_KEY.EMPLOYEE_ID, out1 => #qEKS_DATA_2)
   END_RUNG wire#w1
   // the same network as SCL:
   IF "DB_EKS".HMI.WRITE_NEW_KEY_LEVEL THEN
       #qEKS_START_ADDRESS := 0;
       #qEKS_DATA_LENGTH := 4;
       #qEKS_DATA_1 := "DB_EKS".INSERTED_KEY.LEVEL;
   END_IF;
   IF "DB_EKS".HMI.WRITE_NEW_KEY_ID THEN
       #qEKS_START_ADDRESS := 20;
       #qEKS_DATA_LENGTH := 4;
       #qEKS_DATA_2 := "DB_EKS".INSERTED_KEY.EMPLOYEE_ID;
   END_IF;
   #qEKS_WRITE_CMD := "DB_EKS".HMI.WRITE_NEW_KEY_LEVEL OR "DB_EKS".HMI.WRITE_NEW_KEY_ID;
END_REGION

REGION Network 37: Write Level and Employer ID on Key
   RUNG wire#powerrail
      Contact( "LOG1" )
      wire#w1
      Contact( "DB_EKS".HMI.WRITE_NEW_KEY_LEVEL )
      Contact( #iEKS_JOB_FINISHED )
      R_Coil( "DB_EKS".HMI.WRITE_NEW_KEY_LEVEL )
   END_RUNG
   RUNG wire#w1
      Contact( "DB_EKS".HMI.WRITE_NEW_KEY_ID )
      Contact( #iEKS_JOB_FINISHED )
      R_Coil( "DB_EKS".HMI.WRITE_NEW_KEY_ID )
   END_RUNG
   // the same network as SCL:
   IF "LOG1" AND "DB_EKS".HMI.WRITE_NEW_KEY_LEVEL AND #iEKS_JOB_FINISHED THEN
       "DB_EKS".HMI.WRITE_NEW_KEY_LEVEL := FALSE;
   END_IF;
   IF "LOG1" AND "DB_EKS".HMI.WRITE_NEW_KEY_ID AND #iEKS_JOB_FINISHED THEN
       "DB_EKS".HMI.WRITE_NEW_KEY_ID := FALSE;
   END_IF;
END_REGION
END_FUNCTION
